// SIMATIC S7-200 SMART project (STEP 7-Micro/WIN SMART), CPU ST40

ORGANIZATION_BLOCK MAIN:OB1
TITLE= 
// PROGRAM COMMENTS
// Press F1 for help and example program
//  
BEGIN
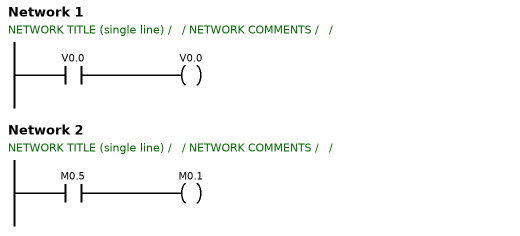
Network 1
// NETWORK TITLE (single line)
//  
// NETWORK COMMENTS
//  
// 
// (network saved uncompiled; LAD cells follow)
// row 0: c0 -| |- V0.0  c1 -( ) V0.0
Network 2
// NETWORK TITLE (single line)
//  
// NETWORK COMMENTS
//  
// 
// (network saved uncompiled; LAD cells follow)
// row 0: c0 -| |- M0.5  c1 -( ) M0.1
END_ORGANIZATION_BLOCK
